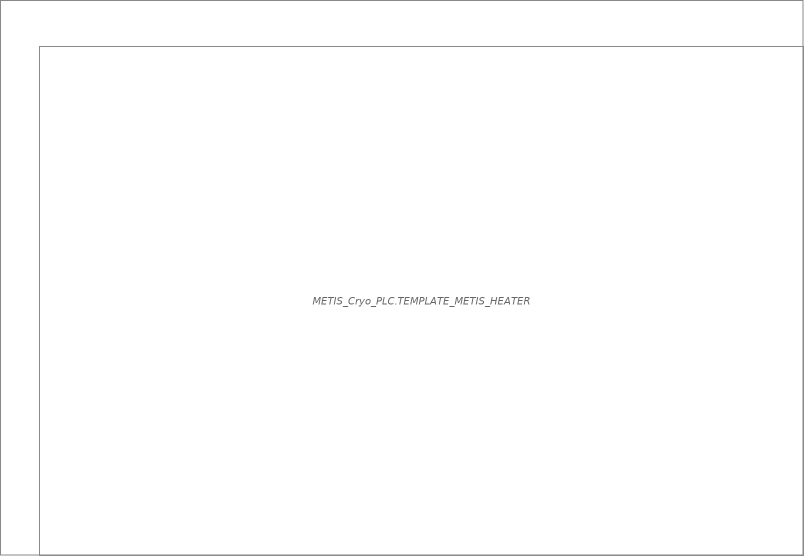
VISUALIZATION VISU_BASE_PLATE_HTR  // 804x556
    Frame (39,46 765x510)
        shows METIS_Cryo_PLC.TEMPLATE_METIS_HEATER(m_instance := MAIN.nott_cryo_ctrl.nott_heaters.h_base_plate)
END_VISUALIZATION

(* stored: Version 1.1.0.1, ProductVersion 3.1.4026.18
   Visu VISU_BASE_PLATE_HTR: Id {81fc91fc-1de6-412d-ae46-a11f0b4841c4} *)
